// TwinCAT 3 PLC project Untitled1
// ProgramVersion: 3.1.4023.0
// libraries:
//   Tc2_Standard, * (Beckhoff Automation GmbH)
//   Tc2_System, * (Beckhoff Automation GmbH)
//   Tc3_Module, * (Beckhoff Automation GmbH)
// project tree:
//   DUTs/ E_ControlMode.TcDUT (not stored), E_PumpControlMode.TcDUT
//   GVLs/ sampleADSGVL.TcGVL (not stored)
//   / PlcTask.TcTTO (not stored)
//   POUs/ MAIN.TcPOU (not stored)
// real-time tasks:
//   TASK PlcTask: cycle T#10ms, priority 20, ADS port 350

// ---- DUTs/E_PumpControlMode.TcDUT
{attribute 'qualified_only'}
{attribute 'strict'}
TYPE E_PumpControlMode :
(
	OFF := 0,					
	CONST_SPEED := 1,				
	CONST_DIFFPRESS := 6,		
	VAR_DIFFPRESS := 7,
	NONE := 99
);
END_TYPE
